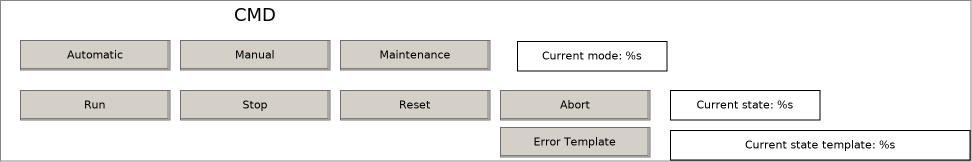
VISUALIZATION VIS_SM  // 972x162
    Button (20,40 150x30), "Automatic"
        tap P_ModeStateManager.bHMIModeRequest_Automatic
    Button (180,40 150x30), "Manual"
        tap P_ModeStateManager.bHMIModeRequest_Manual
    Button (340,40 150x30), "Maintenance"
        tap P_ModeStateManager.bHMIModeRequest_Maintenance
    Label (180,0 150x30), "CMD"
    Rectangle (517,41 150x30), "Current mode: %s", text variable: GVL_Machine.eMode
    Button (20,90 150x30), "Run"
        tap P_ModeStateManager.bHMICommandRequest_Run
    Button (180,90 150x30), "Stop"
        tap P_ModeStateManager.bHMICommandRequest_Stop
    Button (340,90 150x30), "Reset"
        tap P_ModeStateManager.bHMICommandRequest_Reset
    Button (500,90 150x30), "Abort"
        toggle P_ModeStateManager.bHMICommandRequest_Abort
    Rectangle (670,90 150x30), "Current state: %s", text variable: GVL_Machine.eState
    Rectangle (670,130 300x30), "Current state template: %s", text variable: GVL_Machine.eState
    Button (500,127 150x30), "Error Template", colour toggle: P_Template.bError
        toggle P_Template.bError
END_VISUALIZATION

(* stored: Version 1.1.0.1, ProductVersion 3.1.4024.4
   Visu VIS_SM: Id {570f3536-b655-4333-8918-64f711aa2af8} *)
